LIN {X 0,Y 216.618,Z 826.107,A -85,B 0,C 180,E1 3957.922,E2 3957.922} C_VEL
LIN {X 0,Y 210.544,Z 834.012,A -85,B 0,C 180,E1 3957.339,E2 3957.339} C_VEL
LIN {X 0,Y 205.457,Z 840.042,A -85,B 0,C 180,E1 3957.104,E2 3957.104} C_VEL
LIN {X 0,Y 191.375,Z 854.341,A -85,B 0,C 180,E1 3957.411,E2 3957.411} C_VEL
LIN {X 0,Y 185.894,Z 859.552,A -85,B 0,C 180,E1 3957.102,E2 3957.102} C_VEL
LIN {X 0,Y 170.604,Z 873.527,A -85,B 0,C 180,E1 3955.1,E2 3955.1} C_VEL
LIN {X 0,Y 154.315,Z 886.567,A -85,B 0,C 180,E1 3952.467,E2 3952.467} C_VEL
LIN {X 0,Y 137.515,Z 898.345,A -85,B 0,C 180,E1 3948.992,E2 3948.992} C_VEL
LIN {X 0,Y 119.64,Z 909.329,A -85,B 0,C 180,E1 3943.968,E2 3943.968} C_VEL
LIN {X 0,Y 102.455,Z 918.607,A -85,B 0,C 180,E1 3937.022,E2 3937.022} C_VEL
LIN {X 0,Y 86.876,Z 926.217,A -85,B 0,C 180,E1 3927.159,E2 3927.159} C_VEL
LIN {X 0,Y 74.43,Z 932.075,A -85,B 0,C 180,E1 3913.246,E2 3913.246} C_VEL
LIN {X 0,Y 67.439,Z 936.029,A -85,B 0,C 180,E1 3895.465,E2 3895.465} C_VEL
LIN {X 0,Y 66.746,Z 938.029,A -85,B 0,C 180,E1 3877.748,E2 3877.748} C_VEL
LIN {X 0,Y 67.871,Z 938.388,A -85,B 0,C 180,E1 3869.155,E2 3869.155} C_VEL
LIN {X 0,Y 66.823,Z 937.354,A -85,B 0,C 180,E1 3854.374,E2 3854.374} C_VEL
LIN {X 0,Y 71.035,Z 934.386,A -85,B 0,C 180,E1 3835.733,E2 3835.733} C_VEL
LIN {X 0,Y 81.389,Z 929.589,A -85,B 0,C 180,E1 3820.386,E2 3820.386} C_VEL
LIN {X 0,Y 85.695,Z 927.592,A -85,B 0,C 180,E1 3816.255,E2 3816.255} C_VEL
LIN {X 0,Y 73.049,Z 918.736,A -85,B 0,C 180,E1 3770.546,E2 3770.546} C_VEL
LIN {X 0,Y 95.351,Z 912.093,A -85,B 0,C 180,E1 3740.068,E2 3740.068} C_VEL
LIN {X 0,Y 82.095,Z 916.861,A -85,B 0,C 180,E1 3728.402,E2 3728.402} C_VEL
LIN {X 0,Y 72.797,Z 919.826,A -85,B 0,C 180,E1 3713.474,E2 3713.474} C_VEL
LIN {X 0,Y 68.659,Z 921.092,A -85,B 0,C 180,E1 3697.532,E2 3697.532} C_VEL
LIN {X 0,Y 68.75,Z 921.084,A -85,B 0,C 180,E1 3681.638,E2 3681.638} C_VEL
LIN {X 0,Y 73.417,Z 919.686,A -85,B 0,C 180,E1 3665.027,E2 3665.027} C_VEL
LIN {X 0,Y 83.239,Z 916.568,A -85,B 0,C 180,E1 3650.246,E2 3650.246} C_VEL
LIN {X 0,Y 96.56,Z 911.731,A -85,B 0,C 180,E1 3639.047,E2 3639.047} C_VEL
LIN {X 0,Y 111.815,Z 905.264,A -85,B 0,C 180,E1 3630.856,E2 3630.856} C_VEL
LIN {X 0,Y 127.821,Z 897.347,A -85,B 0,C 180,E1 3624.85,E2 3624.85} C_VEL
LIN {X 0,Y 144.067,Z 887.991,A -85,B 0,C 180,E1 3620.305,E2 3620.305} C_VEL
LIN {X 0,Y 159.837,Z 877.473,A -85,B 0,C 180,E1 3616.84,E2 3616.84} C_VEL
LIN {X 0,Y 175.24,Z 865.614,A -85,B 0,C 180,E1 3614.072,E2 3614.072} C_VEL
LIN {X 0,Y 190.012,Z 852.493,A -85,B 0,C 180,E1 3611.826,E2 3611.826} C_VEL
LIN {X 0,Y 204.526,Z 837.542,A -85,B 0,C 180,E1 3609.905,E2 3609.905} C_VEL
LIN {X 0,Y 217.737,Z 821.729,A -85,B 0,C 180,E1 3608.346,E2 3608.346} C_VEL
LIN {X 0,Y 229.709,Z 804.958,A -85,B 0,C 180,E1 3607.046,E2 3607.046} C_VEL
LIN {X 0,Y 240.953,Z 786.217,A -85,B 0,C 180,E1 3605.886,E2 3605.886} C_VEL
LIN {X 0,Y 249.917,Z 768.175,A -85,B 0,C 180,E1 3604.984,E2 3604.984} C_VEL
LIN {X 0,Y 257.662,Z 748.98,A -85,B 0,C 180,E1 3604.195,E2 3604.195} C_VEL
LIN {X 0,Y 264.634,Z 728.339,A -85,B 0,C 180,E1 3603.487,E2 3603.487} C_VEL
LIN {X 0,Y 254.792,Z 756.595,A -85,B 0,C 180,E1 3602.872,E2 3602.872} C_VEL
LIN {X 0,Y 245.665,Z 777.367,A -85,B 0,C 180,E1 3602.267,E2 3602.267} C_VEL
LIN {X 0,Y 235.058,Z 797.078,A -85,B 0,C 180,E1 3601.537,E2 3601.537} C_VEL
LIN {X 0,Y 223.491,Z 815.191,A -85,B 0,C 180,E1 3600.689,E2 3600.689} C_VEL
LIN {X 0,Y 210.689,Z 832.347,A -85,B 0,C 180,E1 3599.633,E2 3599.633} C_VEL
LIN {X 0,Y 196.409,Z 848.853,A -85,B 0,C 180,E1 3598.25,E2 3598.25} C_VEL
LIN {X 0,Y 185.894,Z 859.552,A -85,B 0,C 180,E1 3597.102,E2 3597.102} C_VEL
LIN {X 0,Y 180.234,Z 864.781,A -85,B 0,C 180,E1 3596.749,E2 3596.749} C_VEL
LIN {X 0,Y 164.421,Z 877.238,A -85,B 0,C 180,E1 3596.826,E2 3596.826} C_VEL
LIN {X 0,Y 158.338,Z 881.829,A -85,B 0,C 180,E1 3596.338,E2 3596.338} C_VEL
LIN {X 0,Y 139.96,Z 894.787,A -85,B 0,C 180,E1 3593.231,E2 3593.231} C_VEL
LIN {X 0,Y 121.877,Z 905.816,A -85,B 0,C 180,E1 3589.123,E2 3589.123} C_VEL
LIN {X 0,Y 104.292,Z 915.147,A -85,B 0,C 180,E1 3583.484,E2 3583.484} C_VEL
LIN {X 0,Y 87.099,Z 923.149,A -85,B 0,C 180,E1 3575.082,E2 3575.082} C_VEL
LIN {X 0,Y 71.823,Z 929.609,A -85,B 0,C 180,E1 3562.226,E2 3562.226} C_VEL
LIN {X 0,Y 61.693,Z 934.058,A -85,B 0,C 180,E1 3544.559,E2 3544.559} C_VEL
LIN {X 0,Y 58.442,Z 936.624,A -85,B 0,C 180,E1 3523.858,E2 3523.858} C_VEL
LIN {X 0,Y 59.907,Z 937.393,A -85,B 0,C 180,E1 3509.521,E2 3509.521} C_VEL
LIN {X 0,Y 59.056,Z 936.255,A -85,B 0,C 180,E1 3491.468,E2 3491.468} C_VEL
LIN {X 0,Y 64.789,Z 933.168,A -85,B 0,C 180,E1 3470.746,E2 3470.746} C_VEL
LIN {X 0,Y 76.025,Z 928.598,A -85,B 0,C 180,E1 3455.79,E2 3455.79} C_VEL
LIN {X 0,Y 65.603,Z 920.585,A -85,B 0,C 180,E1 3408.572,E2 3408.572} C_VEL
LIN {X 0,Y 84.945,Z 915.027,A -85,B 0,C 180,E1 3380.181,E2 3380.181} C_VEL
LIN {X 0,Y 71.674,Z 919.179,A -85,B 0,C 180,E1 3366.862,E2 3366.862} C_VEL
LIN {X 0,Y 63.076,Z 921.525,A -85,B 0,C 180,E1 3349.445,E2 3349.445} C_VEL
LIN {X 0,Y 60.291,Z 922.231,A -85,B 0,C 180,E1 3330.951,E2 3330.951} C_VEL
LIN {X 0,Y 62.548,Z 921.649,A -85,B 0,C 180,E1 3312.319,E2 3312.319} C_VEL
LIN {X 0,Y 70.154,Z 919.62,A -85,B 0,C 180,E1 3295.242,E2 3295.242} C_VEL
LIN {X 0,Y 82.083,Z 916.03,A -85,B 0,C 180,E1 3282.007,E2 3282.007} C_VEL
LIN {X 0,Y 96.938,Z 910.777,A -85,B 0,C 180,E1 3272.242,E2 3272.242} C_VEL
LIN {X 0,Y 113.675,Z 903.742,A -85,B 0,C 180,E1 3265.043,E2 3265.043} C_VEL
LIN {X 0,Y 131.632,Z 894.76,A -85,B 0,C 180,E1 3259.624,E2 3259.624} C_VEL
LIN {X 0,Y 148.59,Z 884.696,A -85,B 0,C 180,E1 3255.789,E2 3255.789} C_VEL
LIN {X 0,Y 165.096,Z 873.242,A -85,B 0,C 180,E1 3252.819,E2 3252.819} C_VEL
LIN {X 0,Y 180.985,Z 860.422,A -85,B 0,C 180,E1 3250.456,E2 3250.456} C_VEL
LIN {X 0,Y 196.146,Z 846.214,A -85,B 0,C 180,E1 3248.526,E2 3248.526} C_VEL
LIN {X 0,Y 210.508,Z 830.508,A -85,B 0,C 180,E1 3246.916,E2 3246.916} C_VEL
LIN {X 0,Y 224.023,Z 813.118,A -85,B 0,C 180,E1 3245.543,E2 3245.543} C_VEL
LIN {X 0,Y 235.191,Z 796.122,A -85,B 0,C 180,E1 3244.477,E2 3244.477} C_VEL
LIN {X 0,Y 241.418,Z 785.307,A -85,B 0,C 180,E1 3243.899,E2 3243.899} C_VEL
LIN {X 0,Y 230.336,Z 804.144,A -85,B 0,C 180,E1 3243.235,E2 3243.235} C_VEL
LIN {X 0,Y 218.169,Z 821.724,A -85,B 0,C 180,E1 3242.415,E2 3242.415} C_VEL
LIN {X 0,Y 204.596,Z 838.546,A -85,B 0,C 180,E1 3241.4,E2 3241.4} C_VEL
LIN {X 0,Y 189.479,Z 854.705,A -85,B 0,C 180,E1 3240.052,E2 3240.052} C_VEL
LIN {X 0,Y 173.747,Z 869.308,A -85,B 0,C 180,E1 3238.351,E2 3238.351} C_VEL
LIN {X 0,Y 158.338,Z 881.829,A -85,B 0,C 180,E1 3236.338,E2 3236.338} C_VEL
LIN {X 0,Y 152.133,Z 886.259,A -85,B 0,C 180,E1 3235.787,E2 3235.787} C_VEL
LIN {X 0,Y 134.855,Z 896.583,A -85,B 0,C 180,E1 3235.479,E2 3235.479} C_VEL
LIN {X 0,Y 128.268,Z 900.289,A -85,B 0,C 180,E1 3234.71,E2 3234.71} C_VEL
LIN {X 0,Y 109.564,Z 910.435,A -85,B 0,C 180,E1 3230.268,E2 3230.268} C_VEL
LIN {X 0,Y 90.674,Z 919.211,A -85,B 0,C 180,E1 3223.611,E2 3223.611} C_VEL
LIN {X 0,Y 73.601,Z 926.094,A -85,B 0,C 180,E1 3213.718,E2 3213.718} C_VEL
LIN {X 0,Y 59.253,Z 931.395,A -85,B 0,C 180,E1 3197.944,E2 3197.944} C_VEL
LIN {X 0,Y 51.274,Z 934.831,A -85,B 0,C 180,E1 3175.404,E2 3175.404} C_VEL
LIN {X 0,Y 51.273,Z 936.254,A -85,B 0,C 180,E1 3153.353,E2 3153.353} C_VEL
LIN {X 0,Y 51.777,Z 936.358,A -85,B 0,C 180,E1 3148.893,E2 3148.893} C_VEL
LIN {X 0,Y 51.37,Z 935.197,A -85,B 0,C 180,E1 3128.294,E2 3128.294} C_VEL
LIN {X 0,Y 58.632,Z 932.116,A -85,B 0,C 180,E1 3105.636,E2 3105.636} C_VEL
LIN {X 0,Y 66.259,Z 929.376,A -85,B 0,C 180,E1 3095.281,E2 3095.281} C_VEL
LIN {X 0,Y 58.202,Z 922.188,A -85,B 0,C 180,E1 3046.083,E2 3046.083} C_VEL
LIN {X 0,Y 74.346,Z 917.75,A -85,B 0,C 180,E1 3020.223,E2 3020.223} C_VEL
LIN {X 0,Y 61.243,Z 921.207,A -85,B 0,C 180,E1 3004.851,E2 3004.851} C_VEL
LIN {X 0,Y 53.814,Z 922.891,A -85,B 0,C 180,E1 2985.078,E2 2985.078} C_VEL
LIN {X 0,Y 52.524,Z 923.167,A -85,B 0,C 180,E1 2964.539,E2 2964.539} C_VEL
LIN {X 0,Y 56.954,Z 922.221,A -85,B 0,C 180,E1 2943.967,E2 2943.967} C_VEL
LIN {X 0,Y 67.168,Z 919.768,A -85,B 0,C 180,E1 2926.783,E2 2926.783} C_VEL
LIN {X 0,Y 81.303,Z 915.72,A -85,B 0,C 180,E1 2914.515,E2 2914.515} C_VEL
LIN {X 0,Y 97.815,Z 909.974,A -85,B 0,C 180,E1 2905.9,E2 2905.9} C_VEL
LIN {X 0,Y 114.89,Z 902.803,A -85,B 0,C 180,E1 2899.961,E2 2899.961} C_VEL
LIN {X 0,Y 132.802,Z 893.809,A -85,B 0,C 180,E1 2895.479,E2 2895.479} C_VEL
LIN {X 0,Y 150.347,Z 883.363,A -85,B 0,C 180,E1 2892.142,E2 2892.142} C_VEL
LIN {X 0,Y 167.306,Z 871.497,A -85,B 0,C 180,E1 2889.562,E2 2889.562} C_VEL
LIN {X 0,Y 183.552,Z 858.193,A -85,B 0,C 180,E1 2887.505,E2 2887.505} C_VEL
LIN {X 0,Y 199.003,Z 843.417,A -85,B 0,C 180,E1 2885.817,E2 2885.817} C_VEL
LIN {X 0,Y 213.118,Z 827.652,A -85,B 0,C 180,E1 2884.449,E2 2884.449} C_VEL
LIN {X 0,Y 214.341,Z 826.119,A -85,B 0,C 180,E1 2884.317,E2 2884.317} C_VEL
LIN {X 0,Y 200.329,Z 842.5,A -85,B 0,C 180,E1 2883.393,E2 2883.393} C_VEL
LIN {X 0,Y 184.104,Z 858.875,A -85,B 0,C 180,E1 2882.107,E2 2882.107} C_VEL
LIN {X 0,Y 166.986,Z 873.731,A -85,B 0,C 180,E1 2880.415,E2 2880.415} C_VEL
LIN {X 0,Y 149.058,Z 887.109,A -85,B 0,C 180,E1 2878.179,E2 2878.179} C_VEL
LIN {X 0,Y 130.456,Z 899.041,A -85,B 0,C 180,E1 2875.131,E2 2875.131} C_VEL
LIN {X 0,Y 128.268,Z 900.289,A -85,B 0,C 180,E1 2874.71,E2 2874.71} C_VEL
LIN {X 0,Y 121.603,Z 903.922,A -85,B 0,C 180,E1 2873.828,E2 2873.828} C_VEL
LIN {X 0,Y 103.275,Z 912.023,A -85,B 0,C 180,E1 2872.775,E2 2872.775} C_VEL
LIN {X 0,Y 96.47,Z 914.83,A -85,B 0,C 180,E1 2871.468,E2 2871.468} C_VEL
LIN {X 0,Y 77.923,Z 922.281,A -85,B 0,C 180,E1 2864.234,E2 2864.234} C_VEL
LIN {X 0,Y 60.871,Z 928.153,A -85,B 0,C 180,E1 2852.501,E2 2852.501} C_VEL
LIN {X 0,Y 47.464,Z 932.458,A -85,B 0,C 180,E1 2832.385,E2 2832.385} C_VEL
LIN {X 0,Y 42.535,Z 934.818,A -85,B 0,C 180,E1 2804.985,E2 2804.985} C_VEL
LIN {X 0,Y 43.7,Z 935.34,A -85,B 0,C 180,E1 2788.688,E2 2788.688} C_VEL
LIN {X 0,Y 44.07,Z 934.072,A -85,B 0,C 180,E1 2763.013,E2 2763.013} C_VEL
LIN {X 0,Y 53.64,Z 930.879,A -85,B 0,C 180,E1 2738.471,E2 2738.471} C_VEL
LIN {X 0,Y 56.409,Z 929.95,A -85,B 0,C 180,E1 2734.557,E2 2734.557} C_VEL
LIN {X 0,Y 50.61,Z 923.709,A -85,B 0,C 180,E1 2683.943,E2 2683.943} C_VEL
LIN {X 0,Y 63.763,Z 920.223,A -85,B 0,C 180,E1 2660.404,E2 2660.404} C_VEL
LIN {X 0,Y 50.833,Z 923.026,A -85,B 0,C 180,E1 2642.08,E2 2642.08} C_VEL
LIN {X 0,Y 44.736,Z 924.146,A -85,B 0,C 180,E1 2617.708,E2 2617.708} C_VEL
LIN {X 0,Y 45.931,Z 923.965,A -85,B 0,C 180,E1 2593.561,E2 2593.561} C_VEL
LIN {X 0,Y 53.773,Z 922.515,A -85,B 0,C 180,E1 2572.149,E2 2572.149} C_VEL
LIN {X 0,Y 67.893,Z 919.273,A -85,B 0,C 180,E1 2555.903,E2 2555.903} C_VEL
LIN {X 0,Y 84.388,Z 914.524,A -85,B 0,C 180,E1 2545.777,E2 2545.777} C_VEL
LIN {X 0,Y 102.515,Z 908.022,A -85,B 0,C 180,E1 2538.898,E2 2538.898} C_VEL
LIN {X 0,Y 121.59,Z 899.619,A -85,B 0,C 180,E1 2533.984,E2 2533.984} C_VEL
LIN {X 0,Y 140.319,Z 889.642,A -85,B 0,C 180,E1 2530.465,E2 2530.465} C_VEL
LIN {X 0,Y 157.494,Z 878.775,A -85,B 0,C 180,E1 2527.945,E2 2527.945} C_VEL
LIN {X 0,Y 174.207,Z 866.376,A -85,B 0,C 180,E1 2525.93,E2 2525.93} C_VEL
LIN {X 0,Y 185.336,Z 857.005,A -85,B 0,C 180,E1 2524.749,E2 2524.749} C_VEL
LIN {X 0,Y 168.273,Z 871.741,A -85,B 0,C 180,E1 2523.374,E2 2523.374} C_VEL
LIN {X 0,Y 149.964,Z 885.325,A -85,B 0,C 180,E1 2521.528,E2 2521.528} C_VEL
LIN {X 0,Y 131.006,Z 897.344,A -85,B 0,C 180,E1 2518.987,E2 2518.987} C_VEL
LIN {X 0,Y 111.356,Z 907.927,A -85,B 0,C 180,E1 2515.335,E2 2515.335} C_VEL
LIN {X 0,Y 96.47,Z 914.83,A -85,B 0,C 180,E1 2511.468,E2 2511.468} C_VEL
LIN {X 0,Y 89.643,Z 917.591,A -85,B 0,C 180,E1 2509.941,E2 2509.941} C_VEL
LIN {X 0,Y 70.222,Z 923.445,A -85,B 0,C 180,E1 2506.951,E2 2506.951} C_VEL
LIN {X 0,Y 63.903,Z 925.186,A -85,B 0,C 180,E1 2504.359,E2 2504.359} C_VEL
LIN {X 0,Y 46.757,Z 930.031,A -85,B 0,C 180,E1 2488.802,E2 2488.802} C_VEL
LIN {X 0,Y 36.035,Z 933.05,A -85,B 0,C 180,E1 2461.816,E2 2461.816} C_VEL
LIN {X 0,Y 35.58,Z 934.334,A -85,B 0,C 180,E1 2429.999,E2 2429.999} C_VEL
LIN {X 0,Y 35.468,Z 933.562,A -85,B 0,C 180,E1 2406.753,E2 2406.753} C_VEL
LIN {X 0,Y 44.853,Z 930.844,A -85,B 0,C 180,E1 2376.625,E2 2376.625} C_VEL
LIN {X 0,Y 46.757,Z 930.33,A -85,B 0,C 180,E1 2373.486,E2 2373.486} C_VEL
LIN {X 0,Y 47.552,Z 923.711,A -85,B 0,C 180,E1 2309.691,E2 2309.691} C_VEL
LIN {X 0,Y 53.146,Z 922.474,A -85,B 0,C 180,E1 2300.727,E2 2300.727} C_VEL
LIN {X 0,Y 40.493,Z 924.644,A -85,B 0,C 180,E1 2277.981,E2 2277.981} C_VEL
LIN {X 0,Y 36.479,Z 925.25,A -85,B 0,C 180,E1 2250.001,E2 2250.001} C_VEL
LIN {X 0,Y 40.889,Z 924.615,A -85,B 0,C 180,E1 2220.722,E2 2220.722} C_VEL
LIN {X 0,Y 53.712,Z 922.421,A -85,B 0,C 180,E1 2198.57,E2 2198.57} C_VEL
LIN {X 0,Y 70.909,Z 918.501,A -85,B 0,C 180,E1 2185.517,E2 2185.517} C_VEL
LIN {X 0,Y 90.155,Z 912.706,A -85,B 0,C 180,E1 2177.485,E2 2177.485} C_VEL
LIN {X 0,Y 109.524,Z 905.326,A -85,B 0,C 180,E1 2172.355,E2 2172.355} C_VEL
LIN {X 0,Y 128.501,Z 896.448,A -85,B 0,C 180,E1 2168.809,E2 2168.809} C_VEL
LIN {X 0,Y 146.846,Z 886.123,A -85,B 0,C 180,E1 2166.211,E2 2166.211} C_VEL
LIN {X 0,Y 155.279,Z 880.743,A -85,B 0,C 180,E1 2165.172,E2 2165.172} C_VEL
LIN {X 0,Y 136.207,Z 893.162,A -85,B 0,C 180,E1 2163.276,E2 2163.276} C_VEL
LIN {X 0,Y 116.995,Z 903.787,A -85,B 0,C 180,E1 2160.699,E2 2160.699} C_VEL
LIN {X 0,Y 97.136,Z 913.051,A -85,B 0,C 180,E1 2156.845,E2 2156.845} C_VEL
LIN {X 0,Y 77.931,Z 920.515,A -85,B 0,C 180,E1 2151.091,E2 2151.091} C_VEL
LIN {X 0,Y 63.903,Z 925.186,A -85,B 0,C 180,E1 2144.359,E2 2144.359} C_VEL
LIN {X 0,Y 57.212,Z 926.945,A -85,B 0,C 180,E1 2140.977,E2 2140.977} C_VEL
LIN {X 0,Y 37.624,Z 930.341,A -85,B 0,C 180,E1 2129.856,E2 2129.856} C_VEL
LIN {X 0,Y 33.295,Z 931.079,A -85,B 0,C 180,E1 2122.963,E2 2122.963} C_VEL
LIN {X 0,Y 26.655,Z 933.023,A -85,B 0,C 180,E1 2082.751,E2 2082.751} C_VEL
LIN {X 0,Y 27.496,Z 933.296,A -85,B 0,C 180,E1 2067.915,E2 2067.915} C_VEL
LIN {X 0,Y 30.82,Z 931.894,A -85,B 0,C 180,E1 2027.053,E2 2027.053} C_VEL
LIN {X 0,Y 36.864,Z 930.547,A -85,B 0,C 180,E1 2012.023,E2 2012.023} C_VEL
LIN {X 0,Y 40.901,Z 924.79,A -85,B 0,C 180,E1 1944.075,E2 1944.075} C_VEL
LIN {X 0,Y 42.363,Z 924.48,A -85,B 0,C 180,E1 1941.161,E2 1941.161} C_VEL
LIN {X 0,Y 30.673,Z 926,A -85,B 0,C 180,E1 1913.029,E2 1913.029} C_VEL
LIN {X 0,Y 29.071,Z 926.155,A -85,B 0,C 180,E1 1878.092,E2 1878.092} C_VEL
LIN {X 0,Y 38.261,Z 925.075,A -85,B 0,C 180,E1 1845.123,E2 1845.123} C_VEL
LIN {X 0,Y 54.841,Z 922.342,A -85,B 0,C 180,E1 1826.698,E2 1826.698} C_VEL
LIN {X 0,Y 73.265,Z 918.099,A -85,B 0,C 180,E1 1817.191,E2 1817.191} C_VEL
LIN {X 0,Y 92.803,Z 912.143,A -85,B 0,C 180,E1 1811.346,E2 1811.346} C_VEL
LIN {X 0,Y 111.959,Z 904.75,A -85,B 0,C 180,E1 1807.554,E2 1807.554} C_VEL
LIN {X 0,Y 124.586,Z 899.014,A -85,B 0,C 180,E1 1805.625,E2 1805.625} C_VEL
LIN {X 0,Y 104.131,Z 908.971,A -85,B 0,C 180,E1 1803.007,E2 1803.007} C_VEL
LIN {X 0,Y 83.006,Z 917.424,A -85,B 0,C 180,E1 1798.887,E2 1798.887} C_VEL
LIN {X 0,Y 61.652,Z 924.238,A -85,B 0,C 180,E1 1791.616,E2 1791.616} C_VEL
LIN {X 0,Y 42.631,Z 929.047,A -85,B 0,C 180,E1 1777.959,E2 1777.959} C_VEL
LIN {X 0,Y 33.295,Z 931.079,A -85,B 0,C 180,E1 1762.963,E2 1762.963} C_VEL
LIN {X 0,Y 28.594,Z 931.892,A -85,B 0,C 180,E1 1751.455,E2 1751.455} C_VEL
LIN {X 0,Y 23.208,Z 932.353,A -85,B 0,C 180,E1 1733.945,E2 1733.945} C_VEL
LIN {X 0,Y 19.156,Z 932.181,A -85,B 0,C 180,E1 1699.553,E2 1699.553} C_VEL
LIN {X 0,Y 19.639,Z 931.882,A -85,B 0,C 180,E1 1682.691,E2 1682.691} C_VEL
LIN {X 0,Y 27.205,Z 930.505,A -85,B 0,C 180,E1 1649.727,E2 1649.727} C_VEL
LIN {X 0,Y 31.561,Z 926.226,A -85,B 0,C 180,E1 1582.127,E2 1582.127} C_VEL
LIN {X 0,Y 21.138,Z 927.166,A -85,B 0,C 180,E1 1543.683,E2 1543.683} C_VEL
LIN {X 0,Y 24.542,Z 926.922,A -85,B 0,C 180,E1 1495.225,E2 1495.225} C_VEL
LIN {X 0,Y 39.509,Z 925.295,A -85,B 0,C 180,E1 1467.654,E2 1467.654} C_VEL
LIN {X 0,Y 59.082,Z 921.939,A -85,B 0,C 180,E1 1455.282,E2 1455.282} C_VEL
LIN {X 0,Y 79.935,Z 916.787,A -85,B 0,C 180,E1 1448.817,E2 1448.817} C_VEL
LIN {X 0,Y 92.966,Z 912.745,A -85,B 0,C 180,E1 1446.174,E2 1446.174} C_VEL
LIN {X 0,Y 71.692,Z 920.09,A -85,B 0,C 180,E1 1442.398,E2 1442.398} C_VEL
LIN {X 0,Y 50.803,Z 925.709,A -85,B 0,C 180,E1 1435.485,E2 1435.485} C_VEL
LIN {X 0,Y 30.931,Z 929.713,A -85,B 0,C 180,E1 1419.17,E2 1419.17} C_VEL
LIN {X 0,Y 18.967,Z 931.874,A -85,B 0,C 180,E1 1374.942,E2 1374.942} C_VEL
LIN {X 0,Y 19.38,Z 932.272,A -85,B 0,C 180,E1 1347.041,E2 1347.041} C_VEL
LIN {X 0,Y 19.639,Z 931.882,A -85,B 0,C 180,E1 1322.691,E2 1322.691} C_VEL
LIN {X 0,Y 19.714,Z 931.575,A -85,B 0,C 180,E1 1312.391,E2 1312.391} C_VEL
LIN {X 0,Y 18.765,Z 931.02,A -85,B 0,C 180,E1 1299.604,E2 1299.604} C_VEL
LIN {X 0,Y 17.044,Z 930.146,A -85,B 0,C 180,E1 1280.217,E2 1280.217} C_VEL
LIN {X 0,Y 17.297,Z 928.661,A -85,B 0,C 180,E1 1242.801,E2 1242.801} C_VEL
LIN {X 0,Y 20.588,Z 927.773,A -85,B 0,C 180,E1 1224.138,E2 1224.138} C_VEL
LIN {X 0,Y 12.802,Z 928.225,A -85,B 0,C 180,E1 1161.016,E2 1161.016} C_VEL
LIN {X 0,Y 24.887,Z 927.513,A -85,B 0,C 180,E1 1107.887,E2 1107.887} C_VEL
LIN {X 0,Y 44.97,Z 925.165,A -85,B 0,C 180,E1 1091.953,E2 1091.953} C_VEL
LIN {X 0,Y 59.429,Z 922.576,A -85,B 0,C 180,E1 1086.948,E2 1086.948} C_VEL
LIN {X 0,Y 36.995,Z 927.349,A -85,B 0,C 180,E1 1079.919,E2 1079.919} C_VEL
LIN {X 0,Y 16.518,Z 930.278,A -85,B 0,C 180,E1 1055.222,E2 1055.222} C_VEL
LIN {X 0,Y 11.259,Z 931.246,A -85,B 0,C 180,E1 984.902,E2 984.902} C_VEL
LIN {X 0,Y 17.518,Z 930.258,A -85,B 0,C 180,E1 924.452,E2 924.452} C_VEL
LIN {X 0,Y 17.297,Z 928.661,A -85,B 0,C 180,E1 882.801,E2 882.801} C_VEL
LIN {X 0,Y 16.915,Z 928.497,A -85,B 0,C 180,E1 875.764,E2 875.764} C_VEL
LIN {X 0,Y 14.905,Z 928.517,A -85,B 0,C 180,E1 867.282,E2 867.282} C_VEL
LIN {X 0,Y 10.986,Z 928.707,A -85,B 0,C 180,E1 853.829,E2 853.829} C_VEL
LIN {X 0,Y 7.287,Z 929.158,A -85,B 0,C 180,E1 760.449,E2 760.449} C_VEL
LIN {X 0,Y 8.756,Z 929.136,A -85,B 0,C 180,E1 751.503,E2 751.503} C_VEL
LIN {X 0,Y 22.52,Z 928.504,A -85,B 0,C 180,E1 729.223,E2 729.223} C_VEL
LIN {X 0,Y 2.818,Z 930.171,A -85,B 0,C 180,E1 650.768,E2 650.768} C_VEL
LIN {X 0,Y 3.226,Z 930.206,A -85,B 0,C 180,E1 608.424,E2 608.424} C_VEL
LIN {X 0,Y 8.299,Z 929.821,A -85,B 0,C 180,E1 546.919,E2 546.919} C_VEL
LIN {X 0,Y 9.592,Z 929.116,A -85,B 0,C 180,E1 511.656,E2 511.656} C_VEL
LIN {X 0,Y 8.756,Z 929.136,A -85,B 0,C 180,E1 391.503,E2 391.503} C_VEL
LIN {X 0,Y 10.507,Z 931.136,A -85,B 0,C 180,E1 385.383,E2 385.383} C_VEL
LIN {X 0,Y 10.507,Z 1012.5,A -85,B 0,C 180,E1 385.383,E2 385.383} C_VEL
LIN {X 0,Y 10.507,Z 1012.5,A -85,B 0,C 180,E1 385.383,E2 385.383}

QRS_NEXT_CUT()

QRS_NEXT()
QRS_HOME()

END
